FUNCTION_BLOCK FB_ClearOutputBuffer
VAR_INPUT
	OutputBufferAddress				: PVOID;
	SizeOfOutputBuffer				: UDINT;
END_VAR
VAR_OUTPUT
END_VAR
VAR
	NullItem						: BYTE 		:= 0;
END_VAR


MEMSET(OutputBufferAddress,
		NullItem,
		SizeOfOutputBuffer);

END_FUNCTION_BLOCK

(* stored: Version 1.1.0.1, ProductVersion 3.1.4024.3
   POU FB_ClearOutputBuffer: Id {413b5d5d-fe97-428e-94b2-30caf36f72c6}, SpecialFunc None *)
